// TIA Portal V17 export
// export: Created 2024-08-26T21:07:22.156598Z, ExportSetting WithDefaults, DisplayName Totally Integrated Automation Portal, DisplayVersion V17 Update 7, DisplayName TIA Portal Openness, DisplayVersion V17 Update 7, DisplayName TIA Portal Version Control Interface, DisplayVersion V17, DisplayName SINAMICS Startdrive Advanced, DisplayVersion V17 SP2, DisplayName SINAMICS Startdrive G110M, G120, G120C, G120D, G120P, G115D, DisplayVersion V17 SP2, DisplayName SINAMICS Startdrive G130, G150, S120, S150, SINAMICS MV, S210, DisplayVersion V17 SP2, DisplayName STEP 7 Professional, DisplayVersion V17 Update 7, DisplayName STEP 7 Safety, DisplayVersion V17 Update 6, DisplayName WinCC Advanced / Unified PC, DisplayVersion V17 Update 7
VAR_GLOBAL   // PLC tag table "sequenceMemory"
   aa AT %MW24 : Int;
   a_correctas AT %MW32 : Int;
   a_estados AT %MW34 : Int;
   verificacion_estados_A AT %MW44 : Int;
   verificacion_estados_B AT %MW26 : Int;
   b_estados AT %MW36 : Int;
   numberOfCorrectOutputStates AT %MW38 : Int;
   bb AT %MW40 : Int;
   previousStep AT %MW1112 : Int;
   sequenceRestart AT %M89.1 : Bool;
   stationTurnedOffInSequence AT %M1150.1 : Bool;
END_VAR
